(* IEC 61131-3 sources: plc-vscode/tests/st/all/trust-platform/conformance/cases/init_reset/cfm_init_reset_retain_warm_cold_002, 1 file *)

(* ---- program.st ---- *)
PROGRAM Main
VAR RETAIN
    r : INT := 1;
END_VAR
VAR NON_RETAIN
    n : INT := 2;
END_VAR
VAR
    u : INT := 3;
END_VAR
END_PROGRAM
